// TIA Portal V17 export
// export: Created 2023-12-22T15:08:00.5354652Z, ExportSetting WithDefaults, DisplayName Totally Integrated Automation Portal, DisplayVersion V17, DisplayName TIA Portal Openness, DisplayVersion V17, DisplayName TIA Portal Version Control Interface, DisplayVersion V17, DisplayName STEP 7 Professional, DisplayVersion V17, DisplayName STEP 7 Safety, DisplayVersion V17, DisplayName WinCC Advanced, DisplayVersion V17
FUNCTION_BLOCK "Lock"   // FB2, LAD
{ S7_Optimized_Access := 'FALSE' }
VERSION : 0.1
// stored: AutoNumber true, IsIECCheckEnabled false, SetENOAutomatically false, UDAEnableTagReadback false
   VAR DB_SPECIFIC
      lock : Word;
   END_VAR
BEGIN

REGION Network 1: Блокировка по наличию воды
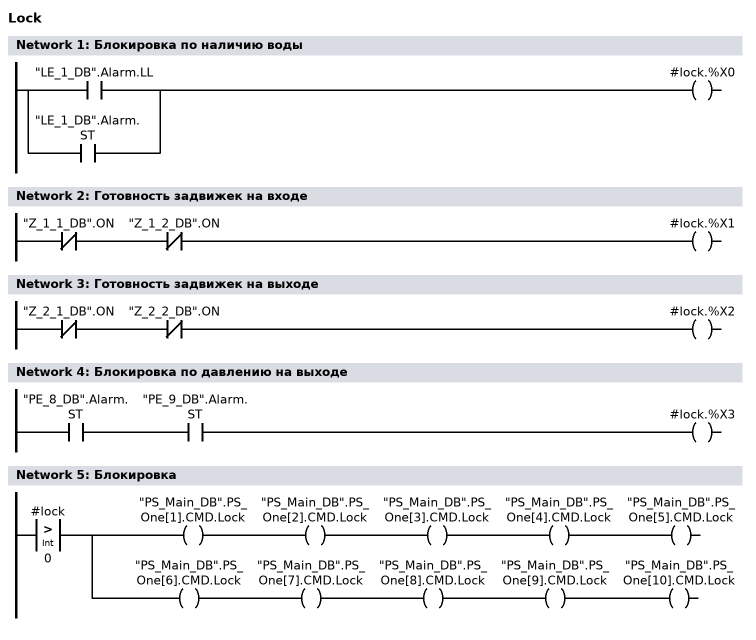
   RUNG wire#powerrail
      Contact( "LE_1_DB".Alarm.LL )
      wire#w1
      Coil( #lock.%X0 )
   END_RUNG
   RUNG wire#powerrail
      Contact( "LE_1_DB".Alarm.ST )
   END_RUNG wire#w1
   // the same network as SCL:
   #lock.%X0 := "LE_1_DB".Alarm.LL OR "LE_1_DB".Alarm.ST;
END_REGION

REGION Network 2: Готовность задвижек на входе
   RUNG wire#powerrail
      I_Contact( "Z_1_1_DB".ON )
      I_Contact( "Z_1_2_DB".ON )
      Coil( #lock.%X1 )
   END_RUNG
   // the same network as SCL:
   #lock.%X1 := NOT "Z_1_1_DB".ON AND NOT "Z_1_2_DB".ON;
END_REGION

REGION Network 3: Готовность задвижек на выходе
   RUNG wire#powerrail
      I_Contact( "Z_2_1_DB".ON )
      I_Contact( "Z_2_2_DB".ON )
      Coil( #lock.%X2 )
   END_RUNG
   // the same network as SCL:
   #lock.%X2 := NOT "Z_2_1_DB".ON AND NOT "Z_2_2_DB".ON;
END_REGION

REGION Network 4: Блокировка по давлению на выходе
   RUNG wire#powerrail
      Contact( "PE_8_DB".Alarm.ST )
      Contact( "PE_9_DB".Alarm.ST )
      Coil( #lock.%X3 )
   END_RUNG
   // the same network as SCL:
   #lock.%X3 := "PE_8_DB".Alarm.ST AND "PE_9_DB".Alarm.ST;
END_REGION

REGION Network 5: Блокировка
   RUNG wire#powerrail
      { S7_Templates := "SrcType := Int" } GT_Contact(in1 := #lock, in2 := 0)
      wire#w1
      Coil( "PS_Main_DB".PS_One[1].CMD.Lock )
      Coil( "PS_Main_DB".PS_One[2].CMD.Lock )
      Coil( "PS_Main_DB".PS_One[3].CMD.Lock )
      Coil( "PS_Main_DB".PS_One[4].CMD.Lock )
      Coil( "PS_Main_DB".PS_One[5].CMD.Lock )
   END_RUNG
   RUNG wire#w1
      Coil( "PS_Main_DB".PS_One[6].CMD.Lock )
      Coil( "PS_Main_DB".PS_One[7].CMD.Lock )
      Coil( "PS_Main_DB".PS_One[8].CMD.Lock )
      Coil( "PS_Main_DB".PS_One[9].CMD.Lock )
      Coil( "PS_Main_DB".PS_One[10].CMD.Lock )
   END_RUNG
   // the same network as SCL:
   "PS_Main_DB".PS_One[1].CMD.Lock := #lock > 0;
   "PS_Main_DB".PS_One[2].CMD.Lock := #lock > 0;
   "PS_Main_DB".PS_One[3].CMD.Lock := #lock > 0;
   "PS_Main_DB".PS_One[4].CMD.Lock := #lock > 0;
   "PS_Main_DB".PS_One[5].CMD.Lock := #lock > 0;
   "PS_Main_DB".PS_One[6].CMD.Lock := #lock > 0;
   "PS_Main_DB".PS_One[7].CMD.Lock := #lock > 0;
   "PS_Main_DB".PS_One[8].CMD.Lock := #lock > 0;
   "PS_Main_DB".PS_One[9].CMD.Lock := #lock > 0;
   "PS_Main_DB".PS_One[10].CMD.Lock := #lock > 0;
END_REGION
END_FUNCTION_BLOCK
